PROGRAM MAIN
VAR
	
END_VAR

P_LightTest();

P_AnalogTest();

P_Safety();

END_PROGRAM

(* stored: Version 1.1.0.1
   POU MAIN: Id {46b1631c-814a-4241-bb42-c62c1f012f3e}, SpecialFunc None *)
